FUNCTION_BLOCK SS3_ifb_Vibrator (* Basic FB with empty ECC *)
  (* Standard: 61499-2 *)
  (* Version 1.0, 2021-08-04, AK121668 *)
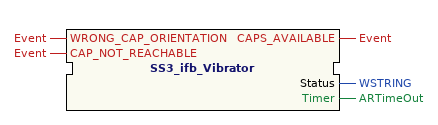
  EVENT_INPUT
    WRONG_CAP_ORIENTATION;
    CAP_NOT_REACHABLE;
  END_EVENT
  EVENT_OUTPUT
    CAPS_AVAILABLE;
  END_EVENT
  VAR_OUTPUT
    Status : WSTRING;
  END_VAR
  PLUGS
    Timer : ARTimeOut;
  END_PLUGS
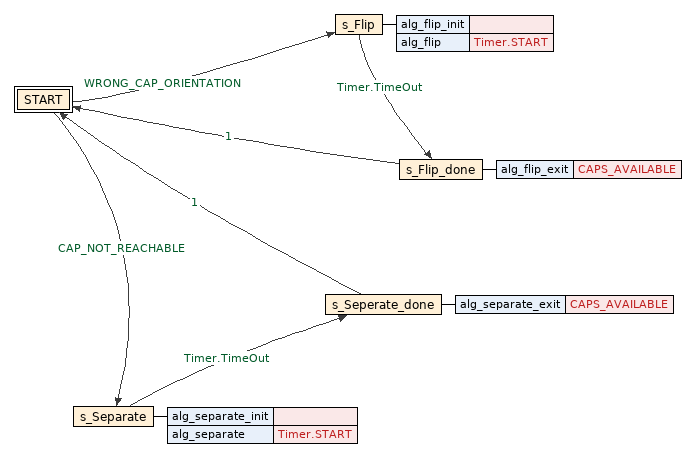
  EC_STATES
    START; (* Initial State *)
    s_Flip : alg_flip_init, alg_flip -> Timer.START;
    s_Separate : alg_separate_init, alg_separate -> Timer.START;
    s_Flip_done : alg_flip_exit -> CAPS_AVAILABLE;
    s_Seperate_done : alg_separate_exit -> CAPS_AVAILABLE;
  END_STATES
  EC_TRANSITIONS
    START TO s_Flip := WRONG_CAP_ORIENTATION;
    START TO s_Separate := CAP_NOT_REACHABLE;
    s_Flip TO s_Flip_done := Timer.TimeOut;
    s_Flip_done TO START := 1;
    s_Separate TO s_Seperate_done := Timer.TimeOut;
    s_Seperate_done TO START := 1;
  END_TRANSITIONS
  ALGORITHM alg_flip_init IN ST:
Timer.DT := T#5s;
Status := "init";
  END_ALGORITHM
  ALGORITHM alg_flip IN ST:
Status := "flipping";
  END_ALGORITHM
  ALGORITHM alg_flip_exit IN ST:
Status := "flipping Done";
  END_ALGORITHM
  ALGORITHM alg_separate_init IN ST:
Timer.DT := T#5s;
Status := "init";
  END_ALGORITHM
  ALGORITHM alg_separate IN ST:
Status := "seperating";
  END_ALGORITHM
  ALGORITHM alg_separate_exit IN ST:
Status := "seperating Done";
  END_ALGORITHM
END_FUNCTION_BLOCK
